// TwinCAT 3 PLC project JsonDOMPLC
// ProgramVersion: 3.1.4024.0
// libraries:
//   Tc2_Standard, * (Beckhoff Automation GmbH)
//   Tc2_System, * (Beckhoff Automation GmbH)
//   Tc2_Utilities, * (Beckhoff Automation GmbH)
//   Tc3_JsonXml, * (Beckhoff Automation GmbH)
//   Tc3_Module, * (Beckhoff Automation GmbH)
// project tree:
//   DUTs/ ST_Machine.TcDUT, ST_MachineState.TcDUT
//   GVLs/ Globals.TcGVL
//   / PlcTask.TcTTO (not stored)
//   POUs/ MAIN.TcPOU
// real-time tasks:
//   TASK PlcTask: cycle T#1ms, priority 20, ADS port 350

// ---- DUTs/ST_Machine.TcDUT
TYPE ST_Machine :
STRUCT
	value : DINT;
END_STRUCT
END_TYPE

// ---- DUTs/ST_MachineState.TcDUT
TYPE ST_MachineState :
STRUCT
	state : DINT;;
END_STRUCT
END_TYPE

// ---- GVLs/Globals.TcGVL
{attribute 'qualified_only'}
VAR_GLOBAL
	machine : ST_MachineState;
END_VAR

// ---- POUs/MAIN.TcPOU
// Damit dieses Beispiel ordnungsgemäß funktioniert muss eine Json-Datei existieren:
// 
// Filename: c:\temp\myJsonContent.json 
//
// File content:
//{
//  "Timestamp":"2017-04-04T12:42:42",
//  "Values": {
//      "Sensor1": 42.41999816894531,
//      "Sensor2": [1,2,3,4,5],
//      "Sensor3": 10
//  }
//}

PROGRAM MAIN
VAR
	fbJson        : FB_JsonDomParser;
	jsonRoot      : SJsonValue;
	jsonProp      : SJsonValue;
	jsonIterator  : SJsonValue;
	jsonIteratorEnd : SJsonValue;
	
	bLoadJson     : BOOL;
	sTimestamp    : STRING;
	fSensor1      : LREAL;
	aSensor2      : ARRAY[0..4] OF DINT;
	nSensor3      : DINT;

	nState 		  : INT := 0;
	bJsonLoaded   : BOOL;

END_VAR

CASE nState OF 

	0:
		bLoadJson := TRUE;
		nState := nState + 1;
	1:
		// Make sure JSON-File exists in specified folder!
		bJsonLoaded := fbJson.LoadDocumentFromFile(sFile := 'c:/temp/myJsonContent.json', bExec:= bLoadJson);	
		// bLoadJsonFile will be set to false when file loading is completed
		IF bLoadJson = FALSE THEN
			IF bJsonLoaded THEN
				// load success
				nState := nState +1;
			ELSE 
				// load failed
				nState := 99;
			END_IF
		END_IF
	2:
		jsonRoot := fbJson.GetDocumentRoot();
		nState := nState +1;
	3:
		jsonProp := fbJson.FindMember(jsonRoot, 'Timestamp');
		IF (jsonProp <> 0) THEN	
  			sTimestamp := fbJson.GetString(jsonProp);
			nState := 100;
		ELSE
			nState := 99;
		END_IF

	99:
		; // Error

	100:
		; // Done
END_CASE

END_PROGRAM
